{attribute 'qualified_only'}
{attribute 'to_string'}
TYPE E_XTS_TRANSPORT_CHECK :
(
  // info for cyclic checks
  INIT_CHECK,
  START_CHECK,    // check cycle start
  XPU_INIT,       // Xpu: initialization


  // errors in fb_TransportUnit.Check()
  POINTER_CHECK           := 9000,
  POINTER_NULL_CTRL,

  POINTER_NULL_STATE,
  POINTER_NULL_XPU_CTRL,

  POINTER_NULL_XPU_STATE,
  POINTER_NULL_XPU_INFO,

  POINTER_NULL_GROUP_ITF,
  POINTER_NULL_GROUP_INFO,

  POINTER_NULL_MOVER,
  POINTER_NULL_MOVER_ITF,

  POINTER_NULL_MOVER_INFO,
  POINTER_NULL_MOVER_LAST_POS,
  POINTER_NULL_MOVER_LAST_GAP,

  POINTER_NULL_STATION_START,
  POINTER_NULL_STATION_ITF,
  POINTER_NULL_STATION_CONTROL,
  POINTER_NULL_STATION_STATE,
  POINTER_NULL_STATION_CTRL_ITF,

  DONE_CHECK              := 10000
)UINT;
END_TYPE

(* stored: Version 1.1.0.1, ProductVersion 3.1.4026.20
   DUT E_XTS_TRANSPORT_CHECK: Id {9f1030d8-dd4b-4a81-a802-58fca891991e} *)
